// TIA Portal V15 export
TagTable "PresetConstants"
  TemplateInt : Int  (1 s, start 4)
